FUNCTION_BLOCK FB_Test3
VAR_INPUT
END_VAR
VAR_OUTPUT
END_VAR
VAR
END_VAR

END_FUNCTION_BLOCK

(* stored: Version 1.1.0.1, ProductVersion 3.1.4024.10
   POU FB_Test3: Id {29b783e8-f2c2-4601-9c30-131f93a571b7}, SpecialFunc None *)
